# EPICS autosave request: tests/testfiles/cfg/SF_SARUN_BPM_OFFS_PV.req
$(SYS):OFFS-X
$(SYS):OFFS-Y
$(SYS):X-REF-FB
$(SYS):Y-REF-FB
